FUNCTION_BLOCK FB_DummyDataReporter IMPLEMENTS I_DataReporter		// Dummy data reporter
	// This will be returned to the caller if no real implementation is found.
	// Methods in this FB will do nothing, thus the project can run happily

METHOD PUBLIC ic_deviceSpeedChanged	// To be called when the (device) speed changes
VAR_INPUT
	iPos:			E_POS;				// Position enumerate
	iMiscArea:		T_SHORT_STR;		// Safety or misc area enumerate (string). If defined/non-empty, use this instead of iPos
	iNew:			INT;				// The new speed value
END_VAR
END_METHOD

METHOD PUBLIC ic_initializeDone	// To be called when a initialization (aka hard reset) is done
VAR_INPUT
	iPos:			E_POS;				// The position
	iMiscArea:		T_SHORT_STR;		// Safety or misc area enumerate (string). If defined/non-empty, use this instead of iPos
	iOrigin:		E_RESET_ORIGIN;
END_VAR
END_METHOD

METHOD PUBLIC ic_operationModeChanged	// To be called when the control signal operation mode changes
VAR_INPUT
	iPos:			E_POS;				// The position
	iMiscArea:		T_SHORT_STR;		// Safety or misc area enumerate (string). If defined/non-empty, use this instead of iPos
	iNew:			E_OPERATION_MODE;	// New operation mode
END_VAR
END_METHOD

METHOD PUBLIC ic_resetDone	// To be called when a reset is done
VAR_INPUT
	iPos:			E_POS;				// The position
	iMiscArea:		T_SHORT_STR;		// Safety or misc area enumerate (string). If defined/non-empty, use this instead of iPos
	iOrigin:		E_RESET_ORIGIN;
	iResetKeyLabel:	T_SHORT_STR;		// What reset key was pressed
END_VAR
END_METHOD

METHOD PUBLIC ic_serviceStateChanged		// To be called when the (control signal) service state changes
VAR_INPUT
	iPos:			E_POS;				// The position
	iMiscArea:		T_SHORT_STR;		// Safety or misc area enumerate (string). If defined/non-empty, use this instead of iPos
	iState:			BOOL;				// TRUE = service activated, FALSE = service deactivated
END_VAR
END_METHOD

END_FUNCTION_BLOCK

(* stored: Version 1.1.0.1, ProductVersion 3.1.4026.18
   POU FB_DummyDataReporter: Id {ae3bd8d0-0d2b-43fa-9328-79a9d09a0685}, SpecialFunc None
   Method ic_deviceSpeedChanged: Id {e3ff05e1-b8fe-4a49-ba3c-531688cea24c}
   Method ic_initializeDone: Id {e6173b74-6923-4a05-b4f0-8eea1d38b03f}
   Method ic_operationModeChanged: Id {ccce60e2-a120-4d25-a30e-55e0f8ddf35f}
   Method ic_resetDone: Id {d6d8eab9-e9ca-402e-a7d4-57afa5b0b0c7}
   Method ic_serviceStateChanged: Id {07eb3339-4b2a-4551-bf3c-05852803fdb9} *)
